FUNCTION_BLOCK StringModel_256000_EX
VAR CONSTANT
	cNumLength:UDINT:=gMaxNumLength;//maximum -+21 4748 3647
	cNumBegin:UDINT:=gNumBegin;
END_VAR
VAR_INPUT
END_VAR
VAR_OUTPUT
	length:UDINT;
	error:BOOL;
	b:ARRAY[cNumBegin..(cNumLength+cNumBegin-1)]OF BYTE;
END_VAR
VAR
	//b:ARRAY[cNumBegin..(cNumLength+cNumBegin-1)]OF BYTE;	
	endPoint:UDINT:=cNumBegin;
END_VAR

(*
	version 1.0 hjm in Zhuhai IA 20171122

	to save string to byte array
*)

METHOD append 
VAR_INPUT
	str:STRING(255);
END_VAR
VAR
	i:INT;
	strTemp:STRING(1);
	_leng:INT;
END_VAR

_leng:=LEN(str);
FOR i:=1 TO _leng DO
	strTemp:=LEFT(str,1);
	str:= DELETE (str,1,1);
	IF endPoint<=cNumLength THEN
		b[endPoint]:=F_ToASC(strTemp);
		endPoint:=endPoint+1;	
	ELSE
		error:=TRUE;
		RETURN;	
	END_IF
END_FOR
length:=endPoint-cNumBegin;
END_METHOD

METHOD getAddr:POINTER TO BYTE;
getAddr:=ADR(b);
END_METHOD

METHOD init 
VAR_INPUT
END_VAR
VAR
	i:UDINT;
END_VAR
FOR i:=cNumBegin TO (cNumLength+cNumBegin-1) DO
	b[i]:=0;
END_FOR
endPoint:=cNumBegin;
error:=FALSE;
END_METHOD

METHOD reset 
VAR_INPUT
END_VAR
endPoint:=cNumBegin;
error:=FALSE;
END_METHOD

END_FUNCTION_BLOCK

(* stored: Version 1.1.0.1, ProductVersion 3.1.4024.4
   POU StringModel_256000_EX: Id {e9efaca8-6831-4f97-92dc-e0d8e6a2f8b7}, SpecialFunc None
   Method append: Id {9655a231-fca8-4d5a-8f88-10a286709c18}
   Method getAddr: Id {707749ba-95de-4bdd-88c9-5385201d3abf}
   Method init: Id {621f7663-3581-400d-afd1-75ef681e0833}
   Method reset: Id {d08ee33a-46f9-495f-8874-1518f9273d52} *)
